INTERFACE PUBLIC I_AnalogInput EXTENDS __System.IQueryInterface

{attribute 'monitoring' := 'call'}
PROPERTY PUBLIC Error : BOOL
GET
END_GET
END_PROPERTY

{attribute 'monitoring' := 'call'}
PROPERTY PUBLIC Overrange : BOOL
GET
END_GET
END_PROPERTY

{attribute 'monitoring' := 'call'}
PROPERTY PUBLIC Underrange : BOOL
GET
END_GET
END_PROPERTY

{attribute 'monitoring' := 'call'}
PROPERTY PUBLIC Value : LREAL
GET
END_GET
END_PROPERTY

END_INTERFACE

(* stored: Version 1.1.0.1, ProductVersion 3.1.4024.12
   Itf I_AnalogInput: Id {0d647588-6d2f-4ac5-9319-c94678430ac7}
   Property Error: Id {67933a15-5b39-4184-827b-503b622c5da0}
   Get Get: Id {145c05f2-afa0-48dc-9ea0-095c9865ccb8}
   Property Overrange: Id {27c23ac9-afa6-4a18-8fc4-94288ef17998}
   Get Get: Id {9c592616-a6df-4261-bf20-b91d1eafa48b}
   Property Underrange: Id {9648cbc1-c6d1-47d5-9520-8874b2ff11c6}
   Get Get: Id {ca00bfbc-a4e7-4898-8580-f4f7912a4d5c}
   Property Value: Id {e5783056-2274-4890-9fbf-391082c99139}
   Get Get: Id {e87217d2-69e6-4be7-8b9a-5d3ebd3b377c} *)
